FUNCTION_BLOCK FB_SDO_WRITE_REAL
VAR_INPUT
	ADSNetID		: STRING(23); 	(* The AMSNetID addresses the EL6751. Can be empty if only one local single channel card is present*)
	PortNr			: WORD; 		(* The Port No. addresses the CANopen Node (see System Manager) *)
	CO_Index		: DWORD; 		(* This is the Index of the CANopen Object Dictionary Entry*)
	CO_SubIndex		: DWORD; 		(* This is the Sub-Index of the CANopen Object Dictionary Entry*)
	StartWriting	: BOOL; 		(* only reset to FALSE after WriteDataFinished=TRUE*)
	WriteData		: REAL; 		(* This real variable contains the data to be written to the CANopen Object Dictionary*)
END_VAR
VAR_OUTPUT
	WriteDataFinished	: BOOL;
	Error			: DWORD;
END_VAR
VAR
	state			: BYTE := 0;
	ADSWRITE		: ADSWRITE;
END_VAR

CASE
state OF
0:
	IF StartWriting THEN
		WriteDataFinished := FALSE;
		Error := 0;
		ADSWrite(
			NETID	:= ADSNetID,
			PORT	:= PortNr,
			IDXGRP	:= CO_Index,
			IDXOFFS	:= CO_SubIndex,
			LEN		:= 4,
			SRCADDR	:= ADR(WriteData),
			WRITE	:= TRUE,
			TMOUT 	:= T#100MS
		);
		IF ADSWrite.err THEN
			state := 2;
			WriteDataFinished := TRUE;
			Error := ADSWrite.ErrId;
		ELSE
			state := 1;
		END_IF
	ELSE
		ADSWrite(
			NETID	:= '',
			PORT	:= PortNr,
			IDXGRP	:= CO_Index,
			IDXOFFS	:= CO_SubIndex,
			LEN		:= 4,
			SRCADDR	:= ADR(WriteData),
			WRITE	:= FALSE,
			TMOUT 	:= T#100MS
		);
	END_IF
	
1:
	ADSWrite(WRITE:= FALSE);
	IF ADSWrite.err THEN
		state := 2;
		WriteDataFinished := TRUE;
		Error := ADSWrite.ErrId;
	ELSE
		IF NOT ADSWrite.busy THEN
			state := 2;
			WriteDataFinished := TRUE;
		END_IF
	END_IF
	
2:
	ADSWrite(WRITE:= FALSE);
	state := 0;
END_CASE

END_FUNCTION_BLOCK

(* stored: Version 1.1.0.1, ProductVersion 3.1.4024.11
   POU FB_SDO_WRITE_REAL: Id {fbd2b633-1518-44e4-802e-bd58bfe27a3f}, SpecialFunc None *)
